FUNCTION_BLOCK FB_HydrolicPump
VAR_INPUT
	mxReset							: BOOL;
	mxEmergency						: BOOL;
	mxAutoMode						: BOOL;
END_VAR
VAR_OUTPUT
(*Errors*)
	Errors							: ST_PumpErrors;
	mxErrorInit						: BOOL;		(* Error, stop immediately. Initialisation neccesary *)
	mxErrorStopinPos				: BOOL;		(* Error, stop in position. Only reset neccesary *)

(* State vars *)
	mxCycleBusy						: BOOL;
	mxInitBusy						: BOOL;
	
(* Vars *)
	mxInitialized					: BOOL;

	
END_VAR
VAR
	ixThermal						AT %I* : BOOL;
	Q								AT %Q* : BOOL;
	
	Hmi_On							: BOOL;
	RT_AutoMode						: R_TRIG;
	SR_ErrorThermal					: SR;
	
END_VAR

Error();

(* Reset hmi when switched to automode*)
RT_AutoMode(CLK:= mxAutoMode);
IF RT_AutoMode.Q THEN Hmi_On:= FALSE; Q:= FALSE; END_IF	

(* Manual control *)
IF NOT mxAutoMode THEN Q:= Hmi_On; END_IF

ACTION Error:
SR_ErrorThermal(SET1:= NOT IxThermal, RESET:= mxReset, Q1=> Errors.Thermal);

(******************************************************************************************************)
mxErrorStopinPos:= FALSE;
mxErrorInit:= Errors.Thermal;
END_ACTION

METHOD M_Init

Q:= FALSE;
END_METHOD

METHOD M_Start : BOOL
VAR_INPUT
END_VAR
Q:=TRUE;

(* Return Value *)
M_Start:= Q;
END_METHOD

METHOD M_Stop : BOOL
VAR_INPUT
END_VAR
Q:= FALSE;

(* Return Value *)
M_Stop:= NOT Q;
END_METHOD

END_FUNCTION_BLOCK

(* stored: Version 1.1.0.1, ProductVersion 3.1.4020.12
   POU FB_HydrolicPump: Id {0ea3798f-f3ef-4b7a-8c69-e34e684e7d45}, SpecialFunc None
   Action Error: Id {37a36703-b1f9-4b3c-a076-ddf7a884235c}
   Method M_Init: Id {8bf75573-5989-4760-bba1-0659b6747b2e}
   Method M_Start: Id {e4d3ab16-c75d-4327-aeb1-b840cda65341}
   Method M_Stop: Id {25eab6d4-a5e3-4d22-be2b-5bfb5d525259} *)
